Fanuc KAREL source: kd00042.KL

PROGRAM KD00042
%STACKSIZE=65535
%PRIORITY=65535
%NOLOCKGROUP
VAR
I : INTEGER
J : INTEGER
B : BOOLEAN
R : REAL
S : STRING[80]
-- UNRESOLVED DECLARATIONS (source type spelling not recovered)
-- N : TYPE_0x1100 (type_u16=0x1100)
BEGIN
I=1
END KD00042
